(* CoDeSys 2.3.9.48 project: test_autoCar.pro *)
(* Libraries: C:\Users\u015329\Documents\Gym_Petershagen\autonomes_Auto\sps\lib\Stepper-03\Stepper_03.lib 10.1.18 07:58:39, Standard.lib 20.5.14 07:13:26, Iecsfc.lib 30.1.13 12:05:12, SYSLIBCALLBACK.LIB 30.1.13 12:05:12 *)

(* PLC configuration (modules and I/O channels)
K-Bus [K_Bus] node 0, in %IB0 out %QB0 {KbusBusMode = 1; KbusCycleTime = 10000; KbusThreadPriority = 0; KbusSetOutputsToZeroOnApplicationStop = 1}
  0750-0673 Steppercontroller [Type_45_1_Channels] node 0, in %IB0 out %QB0
    AT %IB0 [BYTEOnB_I] Status Byte
    AT %IW1 [WORDOnW_I] Actual speed
    AT %IB4 [BYTEOnB_I] Reserved
    AT %IB5 [BYTEOnB_I] Reserved
    AT %IB6 [BYTEOnB_I] Reserved
    AT %IB7 [BYTEOnB_I] Reserved
    AT %IB8 [BYTEOnB_I] Reserved
    AT %IX4.8 [BOOLOnX_I] STOP 1n
    AT %IX4.9 [BOOLOnX_I] REF
    AT %IX4.10 [BOOLOnX_I] positive direction
    AT %IX4.11 [BOOLOnX_I] negative direction
    AT %IX4.12 [BOOLOnX_I] Limit positive direction
    AT %IX4.13 [BOOLOnX_I] Limit negative direction
    AT %IX4.15 [BOOLOnX_I] Reset
    AT %IX5.0 [BOOLOnX_I] ST_ON_TARGET
    AT %IX5.1 [BOOLOnX_I] ST_BUSY
    AT %IX5.2 [BOOLOnX_I] ST_STANDSTILL
    AT %IX5.3 [BOOLOnX_I] ST_VSET
    AT %IX5.4 [BOOLOnX_I] ST_DIRECTION
    AT %IX5.5 [BOOLOnX_I] ST_REF_OK
    AT %IX5.6 [BOOLOnX_I] ST_SETP_M_ACK
    AT %IX5.7 [BOOLOnX_I] ST_ERROR
    AT %IX5.8 [BOOLOnX_I] ST_READY_ACK
    AT %IX5.9 [BOOLOnX_I] ST_STOPn_ACK
    AT %IX5.10 [BOOLOnX_I] ST_START_ACK
    AT %IX5.11 [BOOLOnX_I] ST_SINGLE_ACK
    AT %IX5.12 [BOOLOnX_I] ST_PROGRAM_ACK
    AT %IX5.13 [BOOLOnX_I] ST_REF_ACK
    AT %IX5.14 [BOOLOnX_I] ST_JOG_ACK
    AT %IX5.15 [BOOLOnX_I] ST_MBX_ACK
    AT %QB0 [BYTEOnB_Q] Control byte
    AT %QW1 [WORDOnW_Q] speed
    AT %QW2 [WORDOnW_Q] Acceleration
    AT %QB6 [BYTEOnB_Q] Reserved
    AT %QB7 [BYTEOnB_Q] Reserved
    AT %QB8 [BYTEOnB_Q] Reserved
    AT %QX4.10 [BOOLOnX_Q] drive in positive direction
    AT %QX4.11 [BOOLOnX_Q] drive in negative direction
    AT %QX4.12 [BOOLOnX_Q] Limit positive direction active, only 750-670, 750-671
    AT %QX4.13 [BOOLOnX_Q] Limit negative direction active, only 750-670, 750-671
    AT %QX4.14 [BOOLOnX_Q] choose setup mode
    AT %QX4.15 [BOOLOnX_Q] quit ST_Reset
    AT %QX5.0 [BOOLOnX_Q] Speed divider Bit 0
    AT %QX5.1 [BOOLOnX_Q] Speed divider Bit 1
    AT %QX5.2 [BOOLOnX_Q] CTL ACC FAC BIT0
    AT %QX5.3 [BOOLOnX_Q] CTL ACC FAC BIT1
    AT %QX5.6 [BOOLOnX_Q] Save Value
    AT %QX5.7 [BOOLOnX_Q] Quit Error
    AT %QX5.8 [BOOLOnX_Q] Enable Module
    AT %QX5.9 [BOOLOnX_Q] 0 = stop drive, inverted signal
    AT %QX5.10 [BOOLOnX_Q] 0->1 starts drive
    AT %QX5.11 [BOOLOnX_Q] single positioning, MBX must be inactive
    AT %QX5.12 [BOOLOnX_Q] Program Mode
    AT %QX5.13 [BOOLOnX_Q] Reference Mode
    AT %QX5.14 [BOOLOnX_Q] Jog Mode
    AT %QX5.15 [BOOLOnX_Q] Mailbox Mode
Modbus variables [PFC200MODBUS] node 1, in %IB0 out %QB0 {PlcStopBehaviour = 1; FiledbusErrorBehaviour = 1; TcpOperation = 1; TcpPort = 502; TcpTimeout = 600; UdpOperation = 1; UdpPort = 502; RtuOperation = 0; NodeId = 1; ResponseTimeout = 5000; Interface = 0; Baud = 115200; StopBits = 1; Parity = 1; FlowCtrl = 0; PhysInterface = 0}
Modbus-Master [MB_MASTER] node 2, in %IB0 out %QB0
*)

(* POU PLC_PRG, FBD *)
PROGRAM PLC_PRG
VAR
	Stepper1: MC3_StepperCommunication;
	stepperInputArray	AT %IB0         		: ARRAY [0..11] OF BYTE;
	stepperOutputArray AT %QB0   	       : ARRAY [0..11] OF BYTE;


	Position1: MC3_SetPosition;
	xSetPosition			: BOOL;
	xDoneSetPos			: BOOL;
	xBusySetPos			: BOOL;
	xErrorSetPos			: BOOL;


	Control1: MC3_StepperControlBasic;
	xEnableControl		: BOOL;
	typJobType			: MC3_Mode := MC3_TorqueControl_Edge;
	wModule_673			: WORD := 673;
	xStopStepper			: BOOL;
	iSpeedControl			: INT;
	wAcceleration			: WORD := 1000;
	wDecceleration		: WORD := 1000;
	diTargetPosition		: DINT;
	xStartStepper			: BOOL;
	xErrorReset			: BOOL;
	xDoneControl			: BOOL;
	xBusyControl			: BOOL;
	diCurrentPosition		: DINT;
	iCurrentSpeed		: INT;
	xMailboxActive			: BOOL;
	xErrorControl			: BOOL;
	xWarningControl		: BOOL;
	wStatusControl		: WORD;
	typErrorCodesControl 	: MC3_ERROR_CODES;


	Torque1: MC3_MoveTorque2;
	xEnableTorque		: BOOL;
	iSpeedTorque			: INT;
	wCurrentTorqueProcent	: WORD;
	xDoneTorque			: BOOL;
	xBusyTorque			: BOOL;
END_VAR

VAR CONSTANT
		diZeroPosition		: DINT := 0;
END_VAR
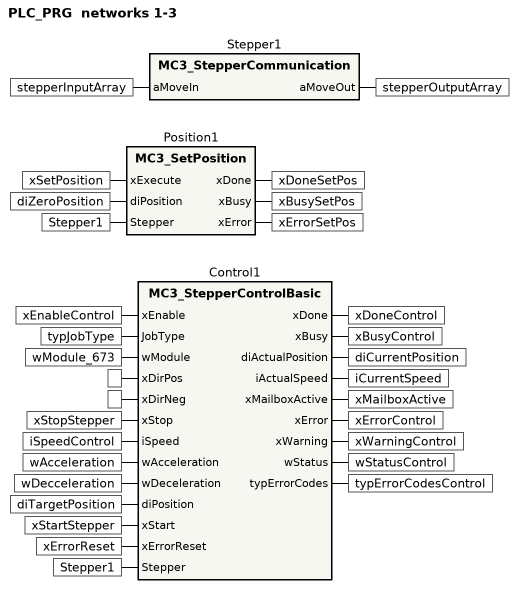
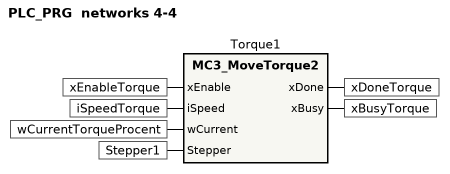
_FBD_ (* Function Block Diagram *)
NETWORK 1
	Stepper1:MC3_StepperCommunication(aMoveIn: stepperInputArray) => stepperOutputArray
NETWORK 2
	Position1:MC3_SetPosition(xExecute: xSetPosition, diPosition: diZeroPosition, Stepper: Stepper1, xBusy => xBusySetPos, xError => xErrorSetPos) => xDoneSetPos
NETWORK 3
	Control1:MC3_StepperControlBasic(xEnable: xEnableControl, JobType: typJobType, wModule: wModule_673, xDirPos: , xDirNeg: , xStop: xStopStepper, iSpeed: iSpeedControl, wAcceleration: wAcceleration, wDeceleration: wDecceleration, diPosition: diTargetPosition, xStart: xStartStepper, xErrorReset: xErrorReset, Stepper: Stepper1, xBusy => xBusyControl, diActualPosition => diCurrentPosition, iActualSpeed => iCurrentSpeed, xMailboxActive => xMailboxActive, xError => xErrorControl, xWarning => xWarningControl, wStatus => wStatusControl, typErrorCodes => typErrorCodesControl) => xDoneControl
NETWORK 4
	Torque1:MC3_MoveTorque2(xEnable: xEnableTorque, iSpeed: iSpeedTorque, wCurrent: wCurrentTorqueProcent, Stepper: Stepper1, xBusy => xBusyTorque) => xDoneTorque
_END_FBD_
(* the same logic as Structured Text *)
(* Network 1 *)
Stepper1(aMoveIn := stepperInputArray);
stepperOutputArray := Stepper1.aMoveOut;
(* Network 2 *)
Position1(xExecute := xSetPosition, diPosition := diZeroPosition, Stepper := Stepper1);
xBusySetPos := Position1.xBusy;
xErrorSetPos := Position1.xError;
xDoneSetPos := Position1.xDone;
(* Network 3: see the listing above *)
(* Network 4 *)
Torque1(xEnable := xEnableTorque, iSpeed := iSpeedTorque, wCurrent := wCurrentTorqueProcent, Stepper := Stepper1);
xBusyTorque := Torque1.xBusy;
xDoneTorque := Torque1.xDone;
END_PROGRAM
